// TIA Portal project "Projekt_skrzyzowanie_ZSP" (V13)

(* hardware
DEVICE "HMI_1"  KTP600 Basic color PN
   slot 0: "HMI"  HMI  6AV6 647-0AD11-3AX0  12.0.0.0
   slot 1: "HMI_RT_1"  KTP600 Basic color PN  6AV6 647-0AD11-3AX0  12.0.0.0
   slot 5: "HMI_1.IE_CP_1"  PROFINET Interface
      slot 1: "PROFINET Interface_1"  PROFINET Interface
         slot 1: "Port_1"  Port
DEVICE "S7-1200 station_2"  S7-1200 Station
   slot 0: "Rack_0"  Rack  V1.0
   slot 1: "PLC_1"  CPU 1212C AC/DC/Rly  6ES7 212-1BD30-0XB0  V2.2
*)

// ===== PLC "PLC_1"  CPU 1212C AC/DC/Rly =====

VAR_GLOBAL   // PLC tag table "Default tag table"
   "Clock_Byte" AT %MB0 : Byte;
   "Clock_10Hz" AT %M0.0 : Bool;
   "Clock_5Hz" AT %M0.1 : Bool;
   "Clock_2.5Hz" AT %M0.2 : Bool;
   "Clock_2Hz" AT %M0.3 : Bool;
   "Clock_1.25Hz" AT %M0.4 : Bool;
   "Clock_1Hz" AT %M0.5 : Bool;
   "Clock_0.625Hz" AT %M0.6 : Bool;
   "Clock_0.5Hz" AT %M0.7 : Bool;
END_VAR

VAR_GLOBAL   // PLC tag table "Tablica_wejsc"
   "przycisk_piesi_1" AT %M10.0 : Bool;
   "przycisk_piesi_2" AT %M10.1 : Bool;
   "przycisk_piesi_3" AT %M10.2 : Bool;
   "przycisk_piesi_4" AT %M10.3 : Bool;
   "przycisk_piesi_5" AT %M10.4 : Bool;
   "przycisk_piesi_6" AT %M10.5 : Bool;
   "petl_ind_czuj_1" AT %I0.0 : Bool;
   "petl_ind_czuj_2" AT %I0.1 : Bool;
   "petl_ind_czuj_3" AT %I0.2 : Bool;
   "petl_ind_czuj_5" AT %I0.3 : Bool;
   "petl_ind_czuj_6" AT %I0.4 : Bool;
   "petl_ind_czuj_8" AT %I0.5 : Bool;
   "petl_ind_czuj_9" AT %I0.6 : Bool;
   "przycisk_trybu_recznego" AT %I0.7 : Bool;
END_VAR

VAR_GLOBAL   // PLC tag table "Tablica_wyjsc"
   "sw_auto_z1" AT %M30.0 : Bool;
   "sw_auto_z2" AT %M30.1 : Bool;
   "sw_auto_z3" AT %M30.2 : Bool;
   "sw_auto_z4" AT %M30.3 : Bool;
   "sw_auto_z5" AT %M30.4 : Bool;
   "sw_auto_z6" AT %M30.5 : Bool;
   "sw_auto_z7" AT %M30.6 : Bool;
   "sw_auto_z8" AT %M30.7 : Bool;
   "sw_auto_z9" AT %M31.0 : Bool;
   "sw_auto_p1" AT %M31.1 : Bool;
   "sw_auto_p2" AT %M31.2 : Bool;
   "sw_auto_p3" AT %M31.3 : Bool;
   "sw_auto_p4" AT %M31.4 : Bool;
   "sw_auto_p5" AT %M31.5 : Bool;
   "sw_auto_p6" AT %M31.6 : Bool;
   "sw_auto_p7" AT %M31.7 : Bool;
   "sw_auto_p8" AT %M32.0 : Bool;
   "sw_auto_p9" AT %M32.1 : Bool;
   "sw_auto_c1" AT %M32.2 : Bool;
   "sw_auto_c2" AT %M32.3 : Bool;
   "sw_auto_c3" AT %M32.4 : Bool;
   "sw_auto_c4" AT %M32.5 : Bool;
   "sw_auto_c5" AT %M32.6 : Bool;
   "sw_auto_c6" AT %M32.7 : Bool;
   "sw_auto_c7" AT %M33.0 : Bool;
   "sw_auto_c8" AT %M33.1 : Bool;
   "sw_auto_c9" AT %M33.2 : Bool;
   "sw_piesi_z1" AT %M33.3 : Bool;
   "sw_piesi_z2" AT %M33.4 : Bool;
   "sw_piesi_z3" AT %M33.5 : Bool;
   "sw_piesi_z4" AT %M33.6 : Bool;
   "sw_piesi_z5" AT %M33.7 : Bool;
   "sw_piesi_z6" AT %M34.0 : Bool;
   "sw_piesi_c1" AT %M34.1 : Bool;
   "sw_piesi_c2" AT %M34.2 : Bool;
   "sw_piesi_c3" AT %M34.3 : Bool;
   "sw_piesi_c4" AT %M34.4 : Bool;
   "sw_piesi_c5" AT %M34.5 : Bool;
   "sw_piesi_c6" AT %M34.6 : Bool;
   "sw_tram_z1" AT %M34.7 : Bool;
   "sw_tram_z2" AT %M35.0 : Bool;
   "sw_tram_c1" AT %M35.1 : Bool;
   "sw_tram_c2" AT %M35.2 : Bool;
END_VAR

VAR_GLOBAL   // PLC tag table "Tablica_zmiennych_programowych"
   "krok_programu" AT %MW20 : Word;
   "tryb_sterowania_recznego" AT %M22.0 : Bool;
   "zmienna_piesi_1" AT %M22.1 : Bool;
   "zmienna_piesi_2" AT %M22.2 : Bool;
   "zmienna_piesi_3" AT %M22.3 : Bool;
   "zmienna_piesi_4" AT %M22.4 : Bool;
   "zmienna_piesi_5" AT %M22.5 : Bool;
   "zmienna_piesi_6" AT %M22.6 : Bool;
   "droga_prioryt_1" AT %M22.7 : Bool;
   "droga_prioryt_2" AT %M23.0 : Bool;
END_VAR

// folder: System blocks/Program resources

DATA_BLOCK "timer_sw_pom_krok_10"   // DB1
{ S7_Optimized_Access := 'FALSE' }
AUTHOR : Simatic
FAMILY : IEC
NAME : IEC_TMR
VERSION : 1.0
// stored: InstanceOfName ?
"?"
BEGIN
END_DATA_BLOCK

DATA_BLOCK "Timer_sw_ziel_krok_11"   // DB2
{ S7_Optimized_Access := 'FALSE' }
AUTHOR : Simatic
FAMILY : IEC
NAME : IEC_TMR
VERSION : 1.0
// stored: InstanceOfName ?
"?"
BEGIN
END_DATA_BLOCK

DATA_BLOCK "Timer_sw_pom_krok_12"   // DB3
{ S7_Optimized_Access := 'FALSE' }
AUTHOR : Simatic
FAMILY : IEC
NAME : IEC_TMR
VERSION : 1.0
// stored: InstanceOfName ?
"?"
BEGIN
END_DATA_BLOCK

DATA_BLOCK "Timer_drogi_priorytetowej_1"   // DB4
{ S7_Optimized_Access := 'FALSE' }
AUTHOR : Simatic
FAMILY : IEC
NAME : IEC_TMR
VERSION : 1.0
// stored: InstanceOfName ?
"?"
BEGIN
END_DATA_BLOCK

DATA_BLOCK "timer_sw_pom_krok_20"   // DB5
{ S7_Optimized_Access := 'FALSE' }
AUTHOR : Simatic
FAMILY : IEC
NAME : IEC_TMR
VERSION : 1.0
// stored: InstanceOfName ?
"?"
BEGIN
END_DATA_BLOCK

DATA_BLOCK "Timer_sw_ziel_krok_21"   // DB6
{ S7_Optimized_Access := 'FALSE' }
AUTHOR : Simatic
FAMILY : IEC
NAME : IEC_TMR
VERSION : 1.0
// stored: InstanceOfName ?
"?"
BEGIN
END_DATA_BLOCK

DATA_BLOCK "Timer_sw_pom_krok_22"   // DB7
{ S7_Optimized_Access := 'FALSE' }
AUTHOR : Simatic
FAMILY : IEC
NAME : IEC_TMR
VERSION : 1.0
// stored: InstanceOfName ?
"?"
BEGIN
END_DATA_BLOCK

DATA_BLOCK "timer_sw_pom_krok_30"   // DB8
{ S7_Optimized_Access := 'FALSE' }
AUTHOR : Simatic
FAMILY : IEC
NAME : IEC_TMR
VERSION : 1.0
// stored: InstanceOfName ?
"?"
BEGIN
END_DATA_BLOCK

DATA_BLOCK "Timer_sw_ziel_krok_31"   // DB9
{ S7_Optimized_Access := 'FALSE' }
AUTHOR : Simatic
FAMILY : IEC
NAME : IEC_TMR
VERSION : 1.0
// stored: InstanceOfName ?
"?"
BEGIN
END_DATA_BLOCK

DATA_BLOCK "Timer_sw_pom_krok_32"   // DB10
{ S7_Optimized_Access := 'FALSE' }
AUTHOR : Simatic
FAMILY : IEC
NAME : IEC_TMR
VERSION : 1.0
// stored: InstanceOfName ?
"?"
BEGIN
END_DATA_BLOCK

DATA_BLOCK "Timer_sw_czer_krok_33"   // DB11
{ S7_Optimized_Access := 'FALSE' }
AUTHOR : Simatic
FAMILY : IEC
NAME : IEC_TMR
VERSION : 1.0
// stored: InstanceOfName ?
"?"
BEGIN
END_DATA_BLOCK

DATA_BLOCK "Timer_sw_czer_krok_13"   // DB12
{ S7_Optimized_Access := 'FALSE' }
AUTHOR : Simatic
FAMILY : IEC
NAME : IEC_TMR
VERSION : 1.0
// stored: InstanceOfName ?
"?"
BEGIN
END_DATA_BLOCK

DATA_BLOCK "Timer_sw_czer_krok_23"   // DB13
{ S7_Optimized_Access := 'FALSE' }
AUTHOR : Simatic
FAMILY : IEC
NAME : IEC_TMR
VERSION : 1.0
// stored: InstanceOfName ?
"?"
BEGIN
END_DATA_BLOCK

DATA_BLOCK "timer_sw_pom_krok_40"   // DB14
{ S7_Optimized_Access := 'FALSE' }
AUTHOR : Simatic
FAMILY : IEC
NAME : IEC_TMR
VERSION : 1.0
// stored: InstanceOfName ?
"?"
BEGIN
END_DATA_BLOCK

DATA_BLOCK "Timer_sw_ziel_krok_41"   // DB15
{ S7_Optimized_Access := 'FALSE' }
AUTHOR : Simatic
FAMILY : IEC
NAME : IEC_TMR
VERSION : 1.0
// stored: InstanceOfName ?
"?"
BEGIN
END_DATA_BLOCK

DATA_BLOCK "Timer_sw_pom_krok_42"   // DB16
{ S7_Optimized_Access := 'FALSE' }
AUTHOR : Simatic
FAMILY : IEC
NAME : IEC_TMR
VERSION : 1.0
// stored: InstanceOfName ?
"?"
BEGIN
END_DATA_BLOCK

DATA_BLOCK "Timer_sw_czer_krok_43"   // DB17
{ S7_Optimized_Access := 'FALSE' }
AUTHOR : Simatic
FAMILY : IEC
NAME : IEC_TMR
VERSION : 1.0
// stored: InstanceOfName ?
"?"
BEGIN
END_DATA_BLOCK

DATA_BLOCK "1Timer_petli_ind_9"   // DB18
{ S7_Optimized_Access := 'FALSE' }
AUTHOR : Simatic
FAMILY : IEC
NAME : IEC_TMR
VERSION : 1.0
// stored: InstanceOfName ?
"?"
BEGIN
END_DATA_BLOCK

DATA_BLOCK "2Timer_petli_ind_9"   // DB19
{ S7_Optimized_Access := 'FALSE' }
AUTHOR : Simatic
FAMILY : IEC
NAME : IEC_TMR
VERSION : 1.0
// stored: InstanceOfName ?
"?"
BEGIN
END_DATA_BLOCK

DATA_BLOCK "Licznik_drog_prior2_1"   // DB20
{ S7_Optimized_Access := 'FALSE' }
AUTHOR : Simatic
FAMILY : IEC
NAME : CNTR
VERSION : 1.0
// stored: InstanceOfName ?
"?"
BEGIN
END_DATA_BLOCK

DATA_BLOCK "Licznik_drog_prior6_1"   // DB21
{ S7_Optimized_Access := 'FALSE' }
AUTHOR : Simatic
FAMILY : IEC
NAME : CNTR
VERSION : 1.0
// stored: InstanceOfName ?
"?"
BEGIN
END_DATA_BLOCK

DATA_BLOCK "Licznik_drog_prior1_2"   // DB22
{ S7_Optimized_Access := 'FALSE' }
AUTHOR : Simatic
FAMILY : IEC
NAME : CNTR
VERSION : 1.0
// stored: InstanceOfName ?
"?"
BEGIN
END_DATA_BLOCK

DATA_BLOCK "Licznik_drog_prior5_2"   // DB23
{ S7_Optimized_Access := 'FALSE' }
AUTHOR : Simatic
FAMILY : IEC
NAME : CNTR
VERSION : 1.0
// stored: InstanceOfName ?
"?"
BEGIN
END_DATA_BLOCK

DATA_BLOCK "Timer_drogi_priorytetowej_2"   // DB24
{ S7_Optimized_Access := 'FALSE' }
AUTHOR : Simatic
FAMILY : IEC
NAME : IEC_TMR
VERSION : 1.0
// stored: InstanceOfName ?
"?"
BEGIN
END_DATA_BLOCK

DATA_BLOCK "1Timer_zmiany_sw_piesi_1"   // DB25
{ S7_Optimized_Access := 'FALSE' }
AUTHOR : Simatic
FAMILY : IEC
NAME : IEC_TMR
VERSION : 1.0
// stored: InstanceOfName ?
"?"
BEGIN
END_DATA_BLOCK

DATA_BLOCK "1Timer_petli_ind_1"   // DB26
{ S7_Optimized_Access := 'FALSE' }
AUTHOR : Simatic
FAMILY : IEC
NAME : IEC_TMR
VERSION : 1.0
// stored: InstanceOfName ?
"?"
BEGIN
END_DATA_BLOCK

DATA_BLOCK "2Timer_petli_ind_1"   // DB27
{ S7_Optimized_Access := 'FALSE' }
AUTHOR : Simatic
FAMILY : IEC
NAME : IEC_TMR
VERSION : 1.0
// stored: InstanceOfName ?
"?"
BEGIN
END_DATA_BLOCK

DATA_BLOCK "1Timer_zmiany_sw_piesi_3"   // DB28
{ S7_Optimized_Access := 'FALSE' }
AUTHOR : Simatic
FAMILY : IEC
NAME : IEC_TMR
VERSION : 1.0
// stored: InstanceOfName ?
"?"
BEGIN
END_DATA_BLOCK

DATA_BLOCK "1Timer_petli_ind_3"   // DB29
{ S7_Optimized_Access := 'FALSE' }
AUTHOR : Simatic
FAMILY : IEC
NAME : IEC_TMR
VERSION : 1.0
// stored: InstanceOfName ?
"?"
BEGIN
END_DATA_BLOCK

DATA_BLOCK "2Timer_petli_ind_3"   // DB30
{ S7_Optimized_Access := 'FALSE' }
AUTHOR : Simatic
FAMILY : IEC
NAME : IEC_TMR
VERSION : 1.0
// stored: InstanceOfName ?
"?"
BEGIN
END_DATA_BLOCK

DATA_BLOCK "1Timer_zmiany_sw_piesi_4"   // DB31
{ S7_Optimized_Access := 'FALSE' }
AUTHOR : Simatic
FAMILY : IEC
NAME : IEC_TMR
VERSION : 1.0
// stored: InstanceOfName ?
"?"
BEGIN
END_DATA_BLOCK

DATA_BLOCK "1Timer_petli_ind_8"   // DB32
{ S7_Optimized_Access := 'FALSE' }
AUTHOR : Simatic
FAMILY : IEC
NAME : IEC_TMR
VERSION : 1.0
// stored: InstanceOfName ?
"?"
BEGIN
END_DATA_BLOCK

DATA_BLOCK "Timer_obsl_petl_ind_1"   // DB33
{ S7_Optimized_Access := 'FALSE' }
AUTHOR : Simatic
FAMILY : IEC
NAME : IEC_TMR
VERSION : 1.0
// stored: InstanceOfName ?
"?"
BEGIN
END_DATA_BLOCK

DATA_BLOCK "Timer_obsl_petl_ind_2"   // DB34
{ S7_Optimized_Access := 'FALSE' }
AUTHOR : Simatic
FAMILY : IEC
NAME : IEC_TMR
VERSION : 1.0
// stored: InstanceOfName ?
"?"
BEGIN
END_DATA_BLOCK

DATA_BLOCK "Timer_obsl_petl_ind_3"   // DB35
{ S7_Optimized_Access := 'FALSE' }
AUTHOR : Simatic
FAMILY : IEC
NAME : IEC_TMR
VERSION : 1.0
// stored: InstanceOfName ?
"?"
BEGIN
END_DATA_BLOCK

DATA_BLOCK "Timer_obsl_petl_ind_4"   // DB36
{ S7_Optimized_Access := 'FALSE' }
AUTHOR : Simatic
FAMILY : IEC
NAME : IEC_TMR
VERSION : 1.0
// stored: InstanceOfName ?
"?"
BEGIN
END_DATA_BLOCK

// folder: (top level)

FUNCTION "Algorytm_glowny" : Void   // FC1, LAD
{ S7_Optimized_Access := 'FALSE' }
VERSION : 0.1
   VAR_TEMP   // added for the SCL form of the ladder/FBD networks
      _w1 : Bool;
   END_VAR
BEGIN

REGION Network 1: Start programu
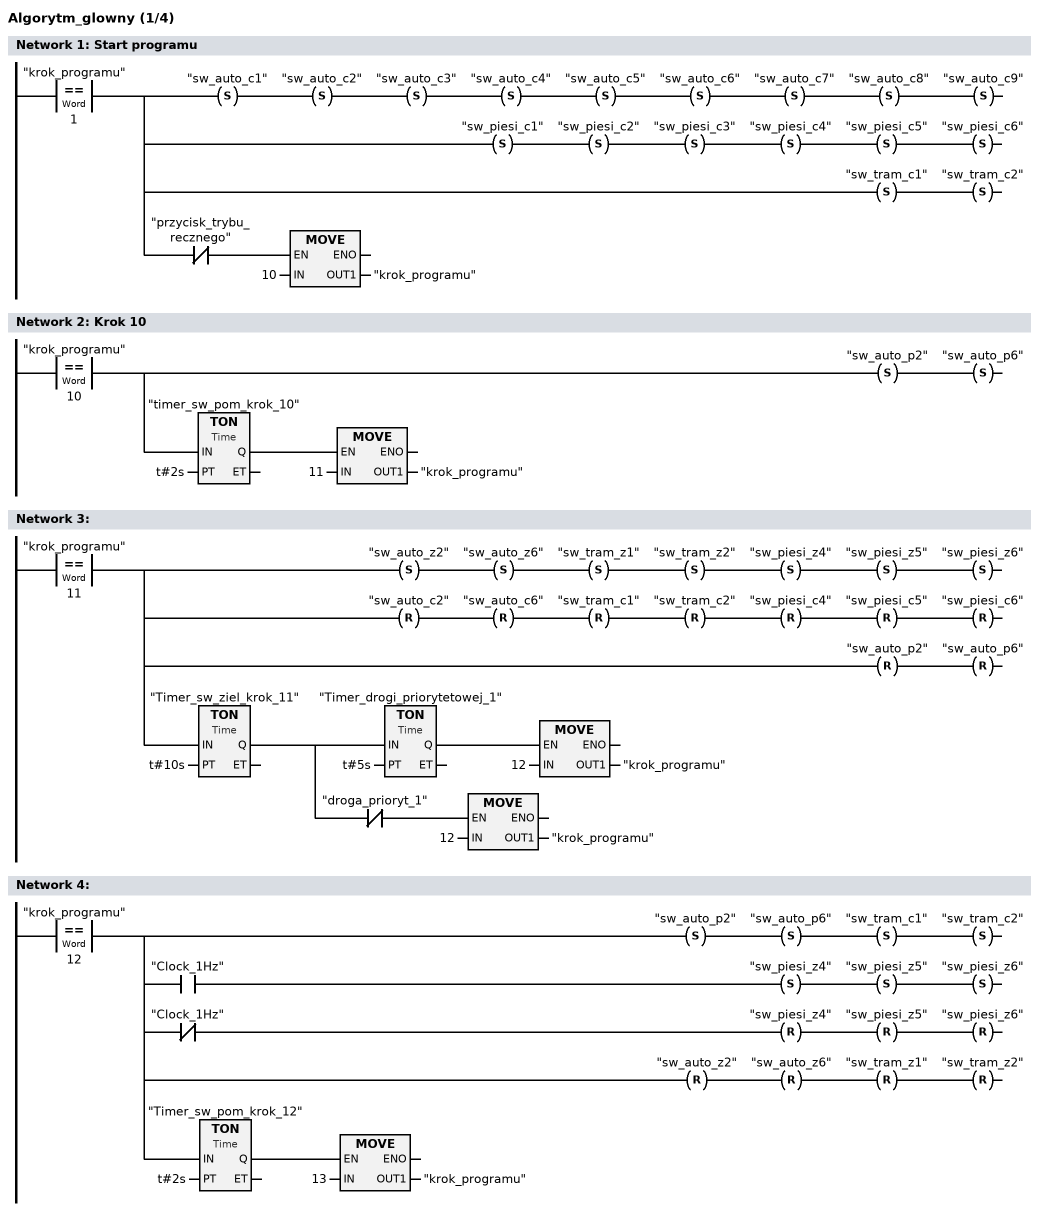
   RUNG wire#powerrail
      { S7_Templates := "SrcType := Word" } EQ_Contact(in1 := "krok_programu", in2 := 1)
      wire#w1
      S_Coil( "sw_auto_c1" )
      S_Coil( "sw_auto_c2" )
      S_Coil( "sw_auto_c3" )
      S_Coil( "sw_auto_c4" )
      S_Coil( "sw_auto_c5" )
      S_Coil( "sw_auto_c6" )
      S_Coil( "sw_auto_c7" )
      S_Coil( "sw_auto_c8" )
      S_Coil( "sw_auto_c9" )
   END_RUNG
   RUNG wire#w1
      S_Coil( "sw_piesi_c1" )
      S_Coil( "sw_piesi_c2" )
      S_Coil( "sw_piesi_c3" )
      S_Coil( "sw_piesi_c4" )
      S_Coil( "sw_piesi_c5" )
      S_Coil( "sw_piesi_c6" )
   END_RUNG
   RUNG wire#w1
      S_Coil( "sw_tram_c1" )
      S_Coil( "sw_tram_c2" )
   END_RUNG
   RUNG wire#w1
      I_Contact( "przycisk_trybu_recznego" )
      Move(in := 10, out1 => "krok_programu")
   END_RUNG
   // the same network as SCL:
   #_w1 := "krok_programu" = 1;
   IF #_w1 THEN
       "sw_auto_c1" := TRUE;
       "sw_auto_c2" := TRUE;
       "sw_auto_c3" := TRUE;
       "sw_auto_c4" := TRUE;
       "sw_auto_c5" := TRUE;
       "sw_auto_c6" := TRUE;
       "sw_auto_c7" := TRUE;
       "sw_auto_c8" := TRUE;
       "sw_auto_c9" := TRUE;
       "sw_piesi_c1" := TRUE;
       "sw_piesi_c2" := TRUE;
       "sw_piesi_c3" := TRUE;
       "sw_piesi_c4" := TRUE;
       "sw_piesi_c5" := TRUE;
       "sw_piesi_c6" := TRUE;
       "sw_tram_c1" := TRUE;
       "sw_tram_c2" := TRUE;
   END_IF;
   IF #_w1 AND NOT "przycisk_trybu_recznego" THEN "krok_programu" := 10; END_IF;
END_REGION

REGION Network 2: Krok 10
   #_w1 := "krok_programu" = 10;
   IF #_w1 THEN
       "sw_auto_p2" := TRUE;
       "sw_auto_p6" := TRUE;
   END_IF;
   "timer_sw_pom_krok_10".TON(IN := #_w1, PT := t#2s);
   IF "timer_sw_pom_krok_10".Q THEN "krok_programu" := 11; END_IF;
END_REGION

REGION Network 3
   #_w1 := "krok_programu" = 11;
   IF #_w1 THEN
       "sw_auto_z2" := TRUE;
       "sw_auto_z6" := TRUE;
       "sw_tram_z1" := TRUE;
       "sw_tram_z2" := TRUE;
       "sw_piesi_z4" := TRUE;
       "sw_piesi_z5" := TRUE;
       "sw_piesi_z6" := TRUE;
       "sw_auto_c2" := FALSE;
       "sw_auto_c6" := FALSE;
       "sw_tram_c1" := FALSE;
       "sw_tram_c2" := FALSE;
       "sw_piesi_c4" := FALSE;
       "sw_piesi_c5" := FALSE;
       "sw_piesi_c6" := FALSE;
       "sw_auto_p2" := FALSE;
       "sw_auto_p6" := FALSE;
   END_IF;
   "Timer_sw_ziel_krok_11".TON(IN := #_w1, PT := t#10s);
   "Timer_drogi_priorytetowej_1".TON(IN := "Timer_sw_ziel_krok_11".Q, PT := t#5s);
   IF "Timer_drogi_priorytetowej_1".Q THEN "krok_programu" := 12; END_IF;
   IF "Timer_sw_ziel_krok_11".Q AND NOT "droga_prioryt_1" THEN "krok_programu" := 12; END_IF;
END_REGION

REGION Network 4
   #_w1 := "krok_programu" = 12;
   IF #_w1 THEN
       "sw_auto_p2" := TRUE;
       "sw_auto_p6" := TRUE;
       "sw_tram_c1" := TRUE;
       "sw_tram_c2" := TRUE;
   END_IF;
   IF #_w1 AND "Clock_1Hz" THEN
       "sw_piesi_z4" := TRUE;
       "sw_piesi_z5" := TRUE;
       "sw_piesi_z6" := TRUE;
   END_IF;
   IF #_w1 AND NOT "Clock_1Hz" THEN
       "sw_piesi_z4" := FALSE;
       "sw_piesi_z5" := FALSE;
       "sw_piesi_z6" := FALSE;
   END_IF;
   IF #_w1 THEN
       "sw_auto_z2" := FALSE;
       "sw_auto_z6" := FALSE;
       "sw_tram_z1" := FALSE;
       "sw_tram_z2" := FALSE;
   END_IF;
   "Timer_sw_pom_krok_12".TON(IN := #_w1, PT := t#2s);
   IF "Timer_sw_pom_krok_12".Q THEN "krok_programu" := 13; END_IF;
END_REGION

REGION Network 5
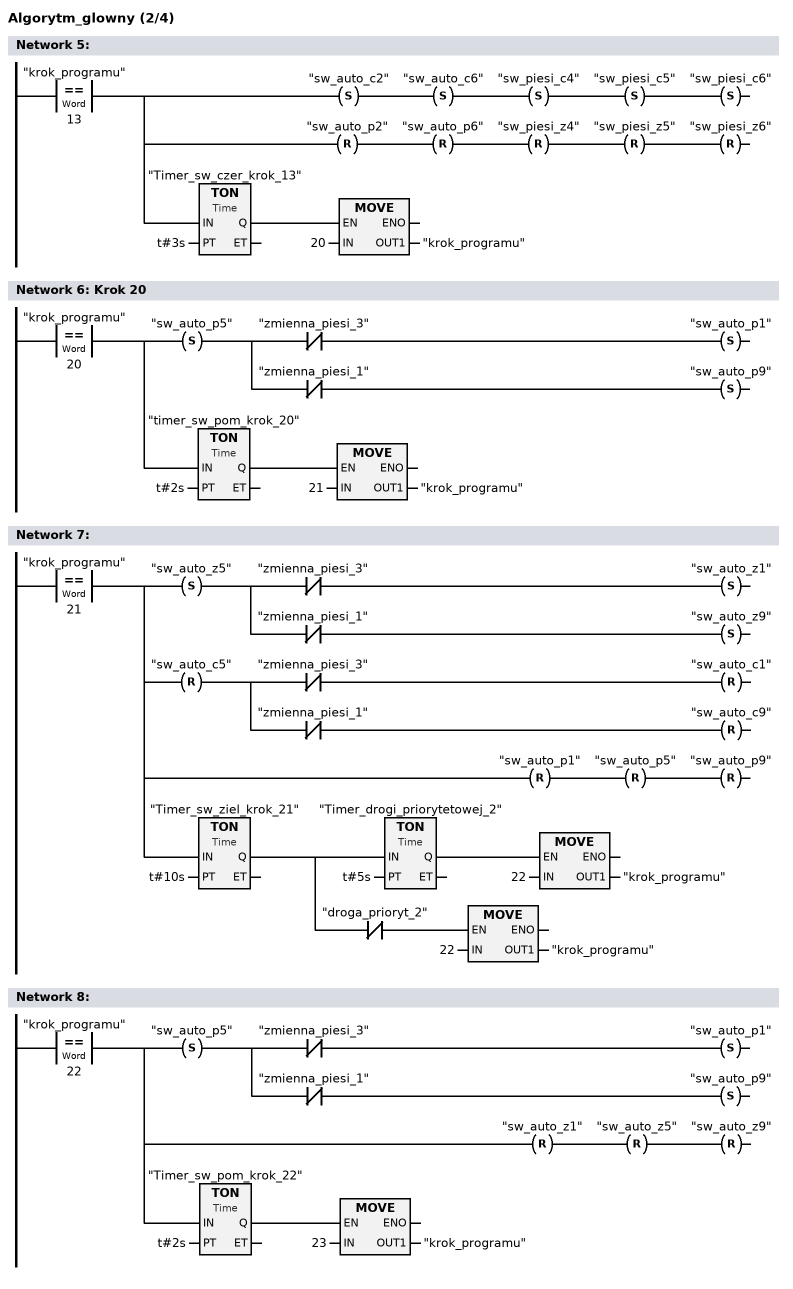
   #_w1 := "krok_programu" = 13;
   IF #_w1 THEN
       "sw_auto_c2" := TRUE;
       "sw_auto_c6" := TRUE;
       "sw_piesi_c4" := TRUE;
       "sw_piesi_c5" := TRUE;
       "sw_piesi_c6" := TRUE;
       "sw_auto_p2" := FALSE;
       "sw_auto_p6" := FALSE;
       "sw_piesi_z4" := FALSE;
       "sw_piesi_z5" := FALSE;
       "sw_piesi_z6" := FALSE;
   END_IF;
   "Timer_sw_czer_krok_13".TON(IN := #_w1, PT := t#3s);
   IF "Timer_sw_czer_krok_13".Q THEN "krok_programu" := 20; END_IF;
END_REGION

REGION Network 6: Krok 20
   #_w1 := "krok_programu" = 20;
   IF #_w1 THEN "sw_auto_p5" := TRUE; END_IF;
   IF #_w1 AND NOT "zmienna_piesi_3" THEN "sw_auto_p1" := TRUE; END_IF;
   IF #_w1 AND NOT "zmienna_piesi_1" THEN "sw_auto_p9" := TRUE; END_IF;
   "timer_sw_pom_krok_20".TON(IN := #_w1, PT := t#2s);
   IF "timer_sw_pom_krok_20".Q THEN "krok_programu" := 21; END_IF;
END_REGION

REGION Network 7
   #_w1 := "krok_programu" = 21;
   IF #_w1 THEN "sw_auto_z5" := TRUE; END_IF;
   IF #_w1 AND NOT "zmienna_piesi_3" THEN "sw_auto_z1" := TRUE; END_IF;
   IF #_w1 AND NOT "zmienna_piesi_1" THEN "sw_auto_z9" := TRUE; END_IF;
   IF #_w1 THEN "sw_auto_c5" := FALSE; END_IF;
   IF #_w1 AND NOT "zmienna_piesi_3" THEN "sw_auto_c1" := FALSE; END_IF;
   IF #_w1 AND NOT "zmienna_piesi_1" THEN "sw_auto_c9" := FALSE; END_IF;
   IF #_w1 THEN
       "sw_auto_p1" := FALSE;
       "sw_auto_p5" := FALSE;
       "sw_auto_p9" := FALSE;
   END_IF;
   "Timer_sw_ziel_krok_21".TON(IN := #_w1, PT := t#10s);
   "Timer_drogi_priorytetowej_2".TON(IN := "Timer_sw_ziel_krok_21".Q, PT := t#5s);
   IF "Timer_drogi_priorytetowej_2".Q THEN "krok_programu" := 22; END_IF;
   IF "Timer_sw_ziel_krok_21".Q AND NOT "droga_prioryt_2" THEN "krok_programu" := 22; END_IF;
END_REGION

REGION Network 8
   #_w1 := "krok_programu" = 22;
   IF #_w1 THEN "sw_auto_p5" := TRUE; END_IF;
   IF #_w1 AND NOT "zmienna_piesi_3" THEN "sw_auto_p1" := TRUE; END_IF;
   IF #_w1 AND NOT "zmienna_piesi_1" THEN "sw_auto_p9" := TRUE; END_IF;
   IF #_w1 THEN
       "sw_auto_z1" := FALSE;
       "sw_auto_z5" := FALSE;
       "sw_auto_z9" := FALSE;
   END_IF;
   "Timer_sw_pom_krok_22".TON(IN := #_w1, PT := t#2s);
   IF "Timer_sw_pom_krok_22".Q THEN "krok_programu" := 23; END_IF;
END_REGION

REGION Network 9
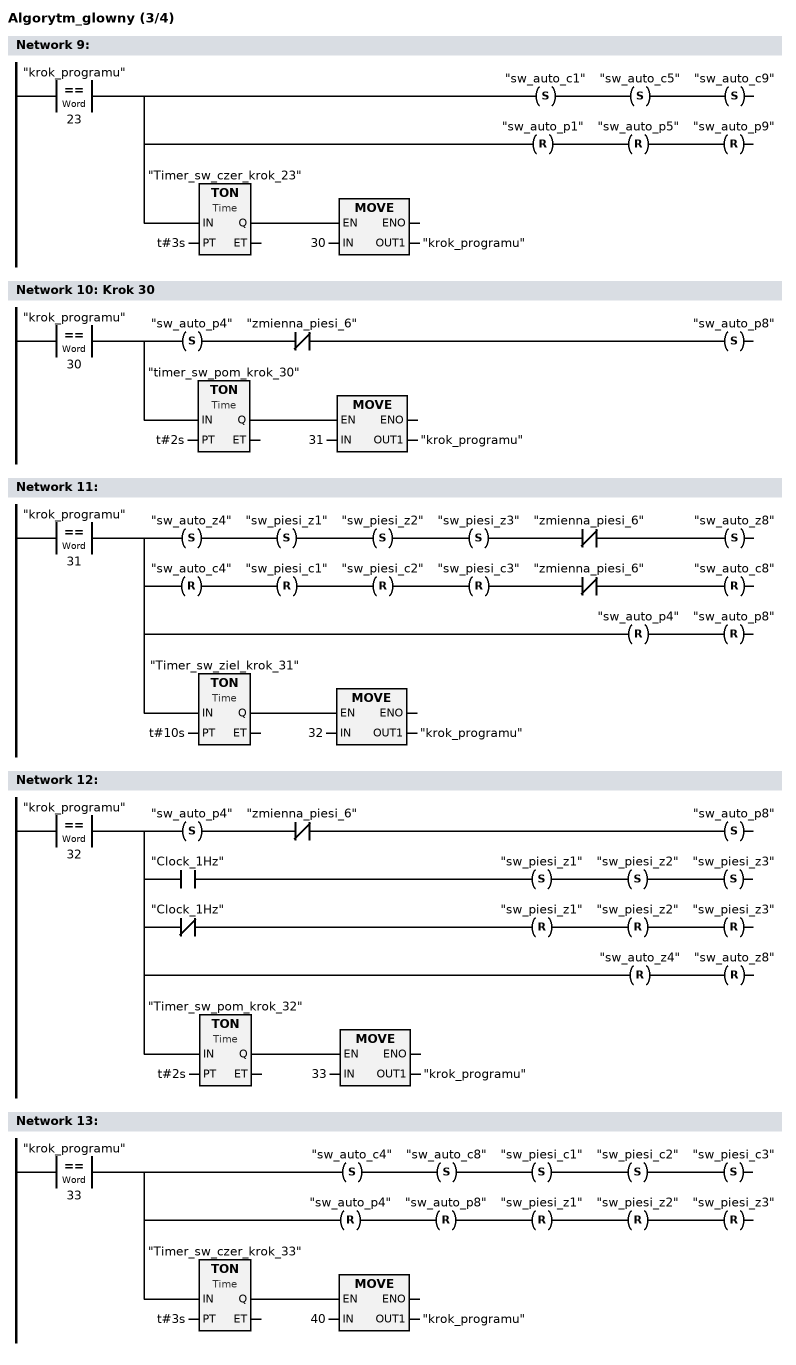
   #_w1 := "krok_programu" = 23;
   IF #_w1 THEN
       "sw_auto_c1" := TRUE;
       "sw_auto_c5" := TRUE;
       "sw_auto_c9" := TRUE;
       "sw_auto_p1" := FALSE;
       "sw_auto_p5" := FALSE;
       "sw_auto_p9" := FALSE;
   END_IF;
   "Timer_sw_czer_krok_23".TON(IN := #_w1, PT := t#3s);
   IF "Timer_sw_czer_krok_23".Q THEN "krok_programu" := 30; END_IF;
END_REGION

REGION Network 10: Krok 30
   #_w1 := "krok_programu" = 30;
   IF #_w1 THEN "sw_auto_p4" := TRUE; END_IF;
   IF #_w1 AND NOT "zmienna_piesi_6" THEN "sw_auto_p8" := TRUE; END_IF;
   "timer_sw_pom_krok_30".TON(IN := #_w1, PT := t#2s);
   IF "timer_sw_pom_krok_30".Q THEN "krok_programu" := 31; END_IF;
END_REGION

REGION Network 11
   #_w1 := "krok_programu" = 31;
   IF #_w1 THEN
       "sw_auto_z4" := TRUE;
       "sw_piesi_z1" := TRUE;
       "sw_piesi_z2" := TRUE;
       "sw_piesi_z3" := TRUE;
   END_IF;
   IF #_w1 AND NOT "zmienna_piesi_6" THEN "sw_auto_z8" := TRUE; END_IF;
   IF #_w1 THEN
       "sw_auto_c4" := FALSE;
       "sw_piesi_c1" := FALSE;
       "sw_piesi_c2" := FALSE;
       "sw_piesi_c3" := FALSE;
   END_IF;
   IF #_w1 AND NOT "zmienna_piesi_6" THEN "sw_auto_c8" := FALSE; END_IF;
   IF #_w1 THEN
       "sw_auto_p4" := FALSE;
       "sw_auto_p8" := FALSE;
   END_IF;
   "Timer_sw_ziel_krok_31".TON(IN := #_w1, PT := t#10s);
   IF "Timer_sw_ziel_krok_31".Q THEN "krok_programu" := 32; END_IF;
END_REGION

REGION Network 12
   #_w1 := "krok_programu" = 32;
   IF #_w1 THEN "sw_auto_p4" := TRUE; END_IF;
   IF #_w1 AND NOT "zmienna_piesi_6" THEN "sw_auto_p8" := TRUE; END_IF;
   IF #_w1 AND "Clock_1Hz" THEN
       "sw_piesi_z1" := TRUE;
       "sw_piesi_z2" := TRUE;
       "sw_piesi_z3" := TRUE;
   END_IF;
   IF #_w1 AND NOT "Clock_1Hz" THEN
       "sw_piesi_z1" := FALSE;
       "sw_piesi_z2" := FALSE;
       "sw_piesi_z3" := FALSE;
   END_IF;
   IF #_w1 THEN
       "sw_auto_z4" := FALSE;
       "sw_auto_z8" := FALSE;
   END_IF;
   "Timer_sw_pom_krok_32".TON(IN := #_w1, PT := t#2s);
   IF "Timer_sw_pom_krok_32".Q THEN "krok_programu" := 33; END_IF;
END_REGION

REGION Network 13
   #_w1 := "krok_programu" = 33;
   IF #_w1 THEN
       "sw_auto_c4" := TRUE;
       "sw_auto_c8" := TRUE;
       "sw_piesi_c1" := TRUE;
       "sw_piesi_c2" := TRUE;
       "sw_piesi_c3" := TRUE;
       "sw_auto_p4" := FALSE;
       "sw_auto_p8" := FALSE;
       "sw_piesi_z1" := FALSE;
       "sw_piesi_z2" := FALSE;
       "sw_piesi_z3" := FALSE;
   END_IF;
   "Timer_sw_czer_krok_33".TON(IN := #_w1, PT := t#3s);
   IF "Timer_sw_czer_krok_33".Q THEN "krok_programu" := 40; END_IF;
END_REGION

REGION Network 14: Krok 40
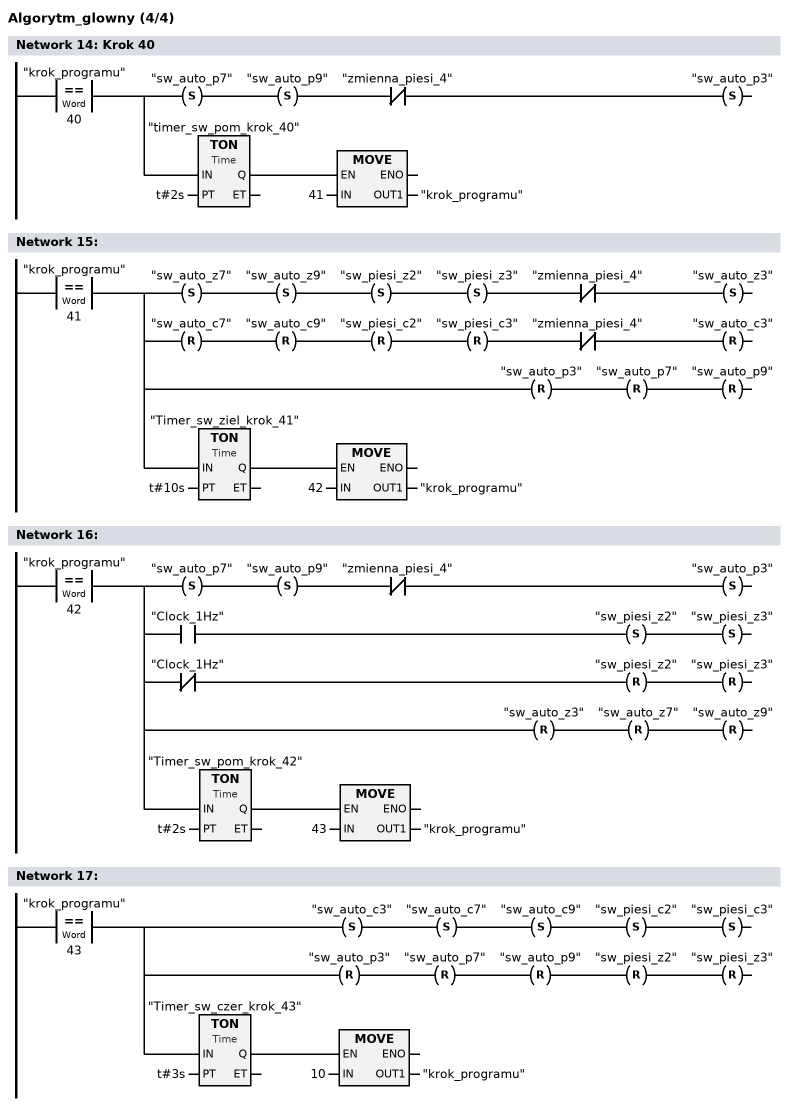
   #_w1 := "krok_programu" = 40;
   IF #_w1 THEN
       "sw_auto_p7" := TRUE;
       "sw_auto_p9" := TRUE;
   END_IF;
   IF #_w1 AND NOT "zmienna_piesi_4" THEN "sw_auto_p3" := TRUE; END_IF;
   "timer_sw_pom_krok_40".TON(IN := #_w1, PT := t#2s);
   IF "timer_sw_pom_krok_40".Q THEN "krok_programu" := 41; END_IF;
END_REGION

REGION Network 15
   #_w1 := "krok_programu" = 41;
   IF #_w1 THEN
       "sw_auto_z7" := TRUE;
       "sw_auto_z9" := TRUE;
       "sw_piesi_z2" := TRUE;
       "sw_piesi_z3" := TRUE;
   END_IF;
   IF #_w1 AND NOT "zmienna_piesi_4" THEN "sw_auto_z3" := TRUE; END_IF;
   IF #_w1 THEN
       "sw_auto_c7" := FALSE;
       "sw_auto_c9" := FALSE;
       "sw_piesi_c2" := FALSE;
       "sw_piesi_c3" := FALSE;
   END_IF;
   IF #_w1 AND NOT "zmienna_piesi_4" THEN "sw_auto_c3" := FALSE; END_IF;
   IF #_w1 THEN
       "sw_auto_p3" := FALSE;
       "sw_auto_p7" := FALSE;
       "sw_auto_p9" := FALSE;
   END_IF;
   "Timer_sw_ziel_krok_41".TON(IN := #_w1, PT := t#10s);
   IF "Timer_sw_ziel_krok_41".Q THEN "krok_programu" := 42; END_IF;
END_REGION

REGION Network 16
   #_w1 := "krok_programu" = 42;
   IF #_w1 THEN
       "sw_auto_p7" := TRUE;
       "sw_auto_p9" := TRUE;
   END_IF;
   IF #_w1 AND NOT "zmienna_piesi_4" THEN "sw_auto_p3" := TRUE; END_IF;
   IF #_w1 AND "Clock_1Hz" THEN
       "sw_piesi_z2" := TRUE;
       "sw_piesi_z3" := TRUE;
   END_IF;
   IF #_w1 AND NOT "Clock_1Hz" THEN
       "sw_piesi_z2" := FALSE;
       "sw_piesi_z3" := FALSE;
   END_IF;
   IF #_w1 THEN
       "sw_auto_z3" := FALSE;
       "sw_auto_z7" := FALSE;
       "sw_auto_z9" := FALSE;
   END_IF;
   "Timer_sw_pom_krok_42".TON(IN := #_w1, PT := t#2s);
   IF "Timer_sw_pom_krok_42".Q THEN "krok_programu" := 43; END_IF;
END_REGION

REGION Network 17
   #_w1 := "krok_programu" = 43;
   IF #_w1 THEN
       "sw_auto_c3" := TRUE;
       "sw_auto_c7" := TRUE;
       "sw_auto_c9" := TRUE;
       "sw_piesi_c2" := TRUE;
       "sw_piesi_c3" := TRUE;
       "sw_auto_p3" := FALSE;
       "sw_auto_p7" := FALSE;
       "sw_auto_p9" := FALSE;
       "sw_piesi_z2" := FALSE;
       "sw_piesi_z3" := FALSE;
   END_IF;
   "Timer_sw_czer_krok_43".TON(IN := #_w1, PT := t#3s);
   IF "Timer_sw_czer_krok_43".Q THEN "krok_programu" := 10; END_IF;
END_REGION
END_FUNCTION

FUNCTION "Sterowanie_reczne" : Void   // FC2, LAD
{ S7_Optimized_Access := 'FALSE' }
VERSION : 0.1
   VAR_TEMP   // added for the SCL form of the ladder/FBD networks
      _w1 : Bool;
   END_VAR
BEGIN

REGION Network 1
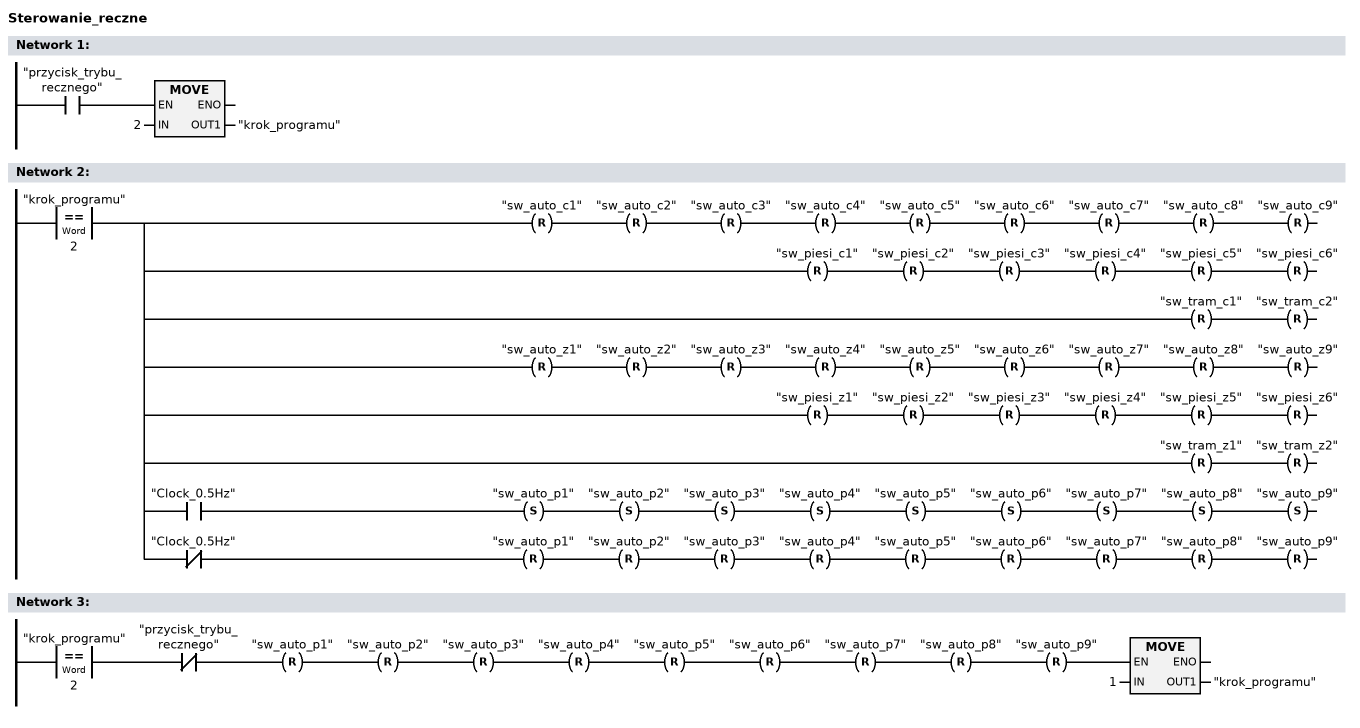
   RUNG wire#powerrail
      Contact( "przycisk_trybu_recznego" )
      Move(in := 2, out1 => "krok_programu")
   END_RUNG
   // the same network as SCL:
   IF "przycisk_trybu_recznego" THEN "krok_programu" := 2; END_IF;
END_REGION

REGION Network 2
   RUNG wire#powerrail
      { S7_Templates := "SrcType := Word" } EQ_Contact(in1 := "krok_programu", in2 := 2)
      wire#w1
      R_Coil( "sw_auto_c1" )
      R_Coil( "sw_auto_c2" )
      R_Coil( "sw_auto_c3" )
      R_Coil( "sw_auto_c4" )
      R_Coil( "sw_auto_c5" )
      R_Coil( "sw_auto_c6" )
      R_Coil( "sw_auto_c7" )
      R_Coil( "sw_auto_c8" )
      R_Coil( "sw_auto_c9" )
   END_RUNG
   RUNG wire#w1
      R_Coil( "sw_piesi_c1" )
      R_Coil( "sw_piesi_c2" )
      R_Coil( "sw_piesi_c3" )
      R_Coil( "sw_piesi_c4" )
      R_Coil( "sw_piesi_c5" )
      R_Coil( "sw_piesi_c6" )
   END_RUNG
   RUNG wire#w1
      R_Coil( "sw_tram_c1" )
      R_Coil( "sw_tram_c2" )
   END_RUNG
   RUNG wire#w1
      R_Coil( "sw_auto_z1" )
      R_Coil( "sw_auto_z2" )
      R_Coil( "sw_auto_z3" )
      R_Coil( "sw_auto_z4" )
      R_Coil( "sw_auto_z5" )
      R_Coil( "sw_auto_z6" )
      R_Coil( "sw_auto_z7" )
      R_Coil( "sw_auto_z8" )
      R_Coil( "sw_auto_z9" )
   END_RUNG
   RUNG wire#w1
      R_Coil( "sw_piesi_z1" )
      R_Coil( "sw_piesi_z2" )
      R_Coil( "sw_piesi_z3" )
      R_Coil( "sw_piesi_z4" )
      R_Coil( "sw_piesi_z5" )
      R_Coil( "sw_piesi_z6" )
   END_RUNG
   RUNG wire#w1
      R_Coil( "sw_tram_z1" )
      R_Coil( "sw_tram_z2" )
   END_RUNG
   RUNG wire#w1
      Contact( "Clock_0.5Hz" )
      S_Coil( "sw_auto_p1" )
      S_Coil( "sw_auto_p2" )
      S_Coil( "sw_auto_p3" )
      S_Coil( "sw_auto_p4" )
      S_Coil( "sw_auto_p5" )
      S_Coil( "sw_auto_p6" )
      S_Coil( "sw_auto_p7" )
      S_Coil( "sw_auto_p8" )
      S_Coil( "sw_auto_p9" )
   END_RUNG
   RUNG wire#w1
      I_Contact( "Clock_0.5Hz" )
      R_Coil( "sw_auto_p1" )
      R_Coil( "sw_auto_p2" )
      R_Coil( "sw_auto_p3" )
      R_Coil( "sw_auto_p4" )
      R_Coil( "sw_auto_p5" )
      R_Coil( "sw_auto_p6" )
      R_Coil( "sw_auto_p7" )
      R_Coil( "sw_auto_p8" )
      R_Coil( "sw_auto_p9" )
   END_RUNG
   // the same network as SCL:
   #_w1 := "krok_programu" = 2;
   IF #_w1 THEN
       "sw_auto_c1" := FALSE;
       "sw_auto_c2" := FALSE;
       "sw_auto_c3" := FALSE;
       "sw_auto_c4" := FALSE;
       "sw_auto_c5" := FALSE;
       "sw_auto_c6" := FALSE;
       "sw_auto_c7" := FALSE;
       "sw_auto_c8" := FALSE;
       "sw_auto_c9" := FALSE;
       "sw_piesi_c1" := FALSE;
       "sw_piesi_c2" := FALSE;
       "sw_piesi_c3" := FALSE;
       "sw_piesi_c4" := FALSE;
       "sw_piesi_c5" := FALSE;
       "sw_piesi_c6" := FALSE;
       "sw_tram_c1" := FALSE;
       "sw_tram_c2" := FALSE;
       "sw_auto_z1" := FALSE;
       "sw_auto_z2" := FALSE;
       "sw_auto_z3" := FALSE;
       "sw_auto_z4" := FALSE;
       "sw_auto_z5" := FALSE;
       "sw_auto_z6" := FALSE;
       "sw_auto_z7" := FALSE;
       "sw_auto_z8" := FALSE;
       "sw_auto_z9" := FALSE;
       "sw_piesi_z1" := FALSE;
       "sw_piesi_z2" := FALSE;
       "sw_piesi_z3" := FALSE;
       "sw_piesi_z4" := FALSE;
       "sw_piesi_z5" := FALSE;
       "sw_piesi_z6" := FALSE;
       "sw_tram_z1" := FALSE;
       "sw_tram_z2" := FALSE;
   END_IF;
   IF #_w1 AND "Clock_0.5Hz" THEN
       "sw_auto_p1" := TRUE;
       "sw_auto_p2" := TRUE;
       "sw_auto_p3" := TRUE;
       "sw_auto_p4" := TRUE;
       "sw_auto_p5" := TRUE;
       "sw_auto_p6" := TRUE;
       "sw_auto_p7" := TRUE;
       "sw_auto_p8" := TRUE;
       "sw_auto_p9" := TRUE;
   END_IF;
   IF #_w1 AND NOT "Clock_0.5Hz" THEN
       "sw_auto_p1" := FALSE;
       "sw_auto_p2" := FALSE;
       "sw_auto_p3" := FALSE;
       "sw_auto_p4" := FALSE;
       "sw_auto_p5" := FALSE;
       "sw_auto_p6" := FALSE;
       "sw_auto_p7" := FALSE;
       "sw_auto_p8" := FALSE;
       "sw_auto_p9" := FALSE;
   END_IF;
END_REGION

REGION Network 3
   RUNG wire#powerrail
      { S7_Templates := "SrcType := Word" } EQ_Contact(in1 := "krok_programu", in2 := 2)
      I_Contact( "przycisk_trybu_recznego" )
      R_Coil( "sw_auto_p1" )
      R_Coil( "sw_auto_p2" )
      R_Coil( "sw_auto_p3" )
      R_Coil( "sw_auto_p4" )
      R_Coil( "sw_auto_p5" )
      R_Coil( "sw_auto_p6" )
      R_Coil( "sw_auto_p7" )
      R_Coil( "sw_auto_p8" )
      R_Coil( "sw_auto_p9" )
      Move(in := 1, out1 => "krok_programu")
   END_RUNG
   // the same network as SCL:
   IF ("krok_programu" = 2) AND NOT "przycisk_trybu_recznego" THEN
       "sw_auto_p1" := FALSE;
       "sw_auto_p2" := FALSE;
       "sw_auto_p3" := FALSE;
       "sw_auto_p4" := FALSE;
       "sw_auto_p5" := FALSE;
       "sw_auto_p6" := FALSE;
       "sw_auto_p7" := FALSE;
       "sw_auto_p8" := FALSE;
       "sw_auto_p9" := FALSE;
       "krok_programu" := 1;
   END_IF;
END_REGION
END_FUNCTION

FUNCTION "Obsluga_drogi_priorytetowej" : Void   // FC3, LAD
{ S7_Optimized_Access := 'FALSE' }
VERSION : 0.1
BEGIN

REGION Network 1
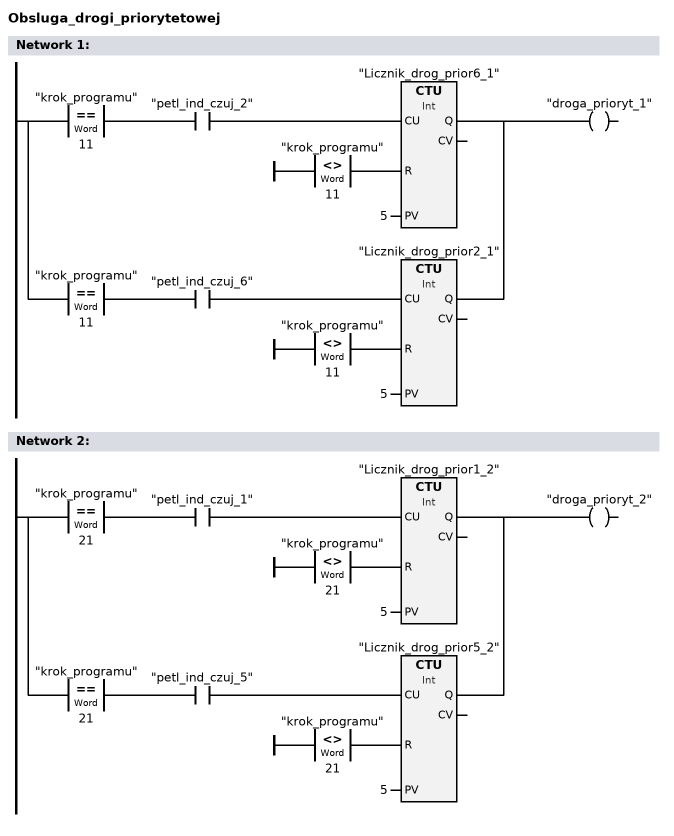
   "Licznik_drog_prior6_1".CTU(CU := ("krok_programu" = 11) AND "petl_ind_czuj_2",
                           R := "krok_programu" <> 11,
                           PV := 5);
   "Licznik_drog_prior2_1".CTU(CU := ("krok_programu" = 11) AND "petl_ind_czuj_6",
                           R := "krok_programu" <> 11,
                           PV := 5);
   "droga_prioryt_1" := "Licznik_drog_prior6_1".Q OR "Licznik_drog_prior2_1".Q;
END_REGION

REGION Network 2
   "Licznik_drog_prior1_2".CTU(CU := ("krok_programu" = 21) AND "petl_ind_czuj_1",
                           R := "krok_programu" <> 21,
                           PV := 5);
   "Licznik_drog_prior5_2".CTU(CU := ("krok_programu" = 21) AND "petl_ind_czuj_5",
                           R := "krok_programu" <> 21,
                           PV := 5);
   "droga_prioryt_2" := "Licznik_drog_prior1_2".Q OR "Licznik_drog_prior5_2".Q;
END_REGION
END_FUNCTION

FUNCTION "Przyciski_pieszych" : Void   // FC4, LAD
{ S7_Optimized_Access := 'FALSE' }
VERSION : 0.1
   VAR_TEMP   // added for the SCL form of the ladder/FBD networks
      _w1 : Bool;
   END_VAR
BEGIN

REGION Network 1: Piesi 1
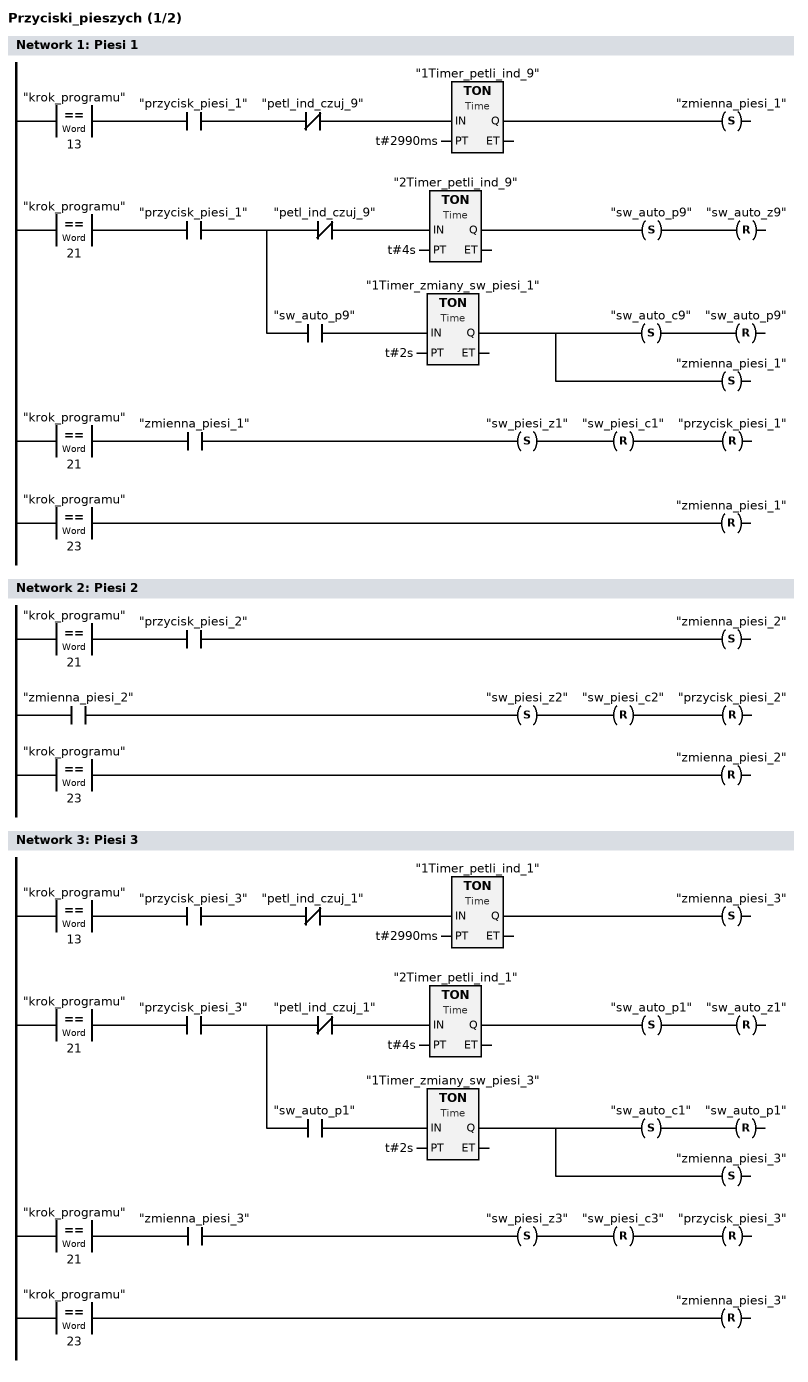
   "1Timer_petli_ind_9".TON(IN := ("krok_programu" = 13) AND "przycisk_piesi_1" AND NOT "petl_ind_czuj_9",
                           PT := t#2990ms);
   IF "1Timer_petli_ind_9".Q THEN "zmienna_piesi_1" := TRUE; END_IF;
   #_w1 := ("krok_programu" = 21) AND "przycisk_piesi_1";
   "2Timer_petli_ind_9".TON(IN := #_w1 AND NOT "petl_ind_czuj_9", PT := t#4s);
   IF "2Timer_petli_ind_9".Q THEN
       "sw_auto_p9" := TRUE;
       "sw_auto_z9" := FALSE;
   END_IF;
   "1Timer_zmiany_sw_piesi_1".TON(IN := #_w1 AND "sw_auto_p9", PT := t#2s);
   IF "1Timer_zmiany_sw_piesi_1".Q THEN
       "sw_auto_c9" := TRUE;
       "sw_auto_p9" := FALSE;
       "zmienna_piesi_1" := TRUE;
   END_IF;
   IF ("krok_programu" = 21) AND "zmienna_piesi_1" THEN
       "sw_piesi_z1" := TRUE;
       "sw_piesi_c1" := FALSE;
       "przycisk_piesi_1" := FALSE;
   END_IF;
   IF "krok_programu" = 23 THEN "zmienna_piesi_1" := FALSE; END_IF;
END_REGION

REGION Network 2: Piesi 2
   RUNG wire#powerrail
      { S7_Templates := "SrcType := Word" } EQ_Contact(in1 := "krok_programu", in2 := 21)
      Contact( "przycisk_piesi_2" )
      S_Coil( "zmienna_piesi_2" )
   END_RUNG
   RUNG wire#powerrail
      Contact( "zmienna_piesi_2" )
      S_Coil( "sw_piesi_z2" )
      R_Coil( "sw_piesi_c2" )
      R_Coil( "przycisk_piesi_2" )
   END_RUNG
   RUNG wire#powerrail
      { S7_Templates := "SrcType := Word" } EQ_Contact(in1 := "krok_programu", in2 := 23)
      R_Coil( "zmienna_piesi_2" )
   END_RUNG
   // the same network as SCL:
   IF ("krok_programu" = 21) AND "przycisk_piesi_2" THEN "zmienna_piesi_2" := TRUE; END_IF;
   IF "zmienna_piesi_2" THEN
       "sw_piesi_z2" := TRUE;
       "sw_piesi_c2" := FALSE;
       "przycisk_piesi_2" := FALSE;
   END_IF;
   IF "krok_programu" = 23 THEN "zmienna_piesi_2" := FALSE; END_IF;
END_REGION

REGION Network 3: Piesi 3
   "1Timer_petli_ind_1".TON(IN := ("krok_programu" = 13) AND "przycisk_piesi_3" AND NOT "petl_ind_czuj_1",
                           PT := t#2990ms);
   IF "1Timer_petli_ind_1".Q THEN "zmienna_piesi_3" := TRUE; END_IF;
   #_w1 := ("krok_programu" = 21) AND "przycisk_piesi_3";
   "2Timer_petli_ind_1".TON(IN := #_w1 AND NOT "petl_ind_czuj_1", PT := t#4s);
   IF "2Timer_petli_ind_1".Q THEN
       "sw_auto_p1" := TRUE;
       "sw_auto_z1" := FALSE;
   END_IF;
   "1Timer_zmiany_sw_piesi_3".TON(IN := #_w1 AND "sw_auto_p1", PT := t#2s);
   IF "1Timer_zmiany_sw_piesi_3".Q THEN
       "sw_auto_c1" := TRUE;
       "sw_auto_p1" := FALSE;
       "zmienna_piesi_3" := TRUE;
   END_IF;
   IF ("krok_programu" = 21) AND "zmienna_piesi_3" THEN
       "sw_piesi_z3" := TRUE;
       "sw_piesi_c3" := FALSE;
       "przycisk_piesi_3" := FALSE;
   END_IF;
   IF "krok_programu" = 23 THEN "zmienna_piesi_3" := FALSE; END_IF;
END_REGION

REGION Network 4: Piesi 4
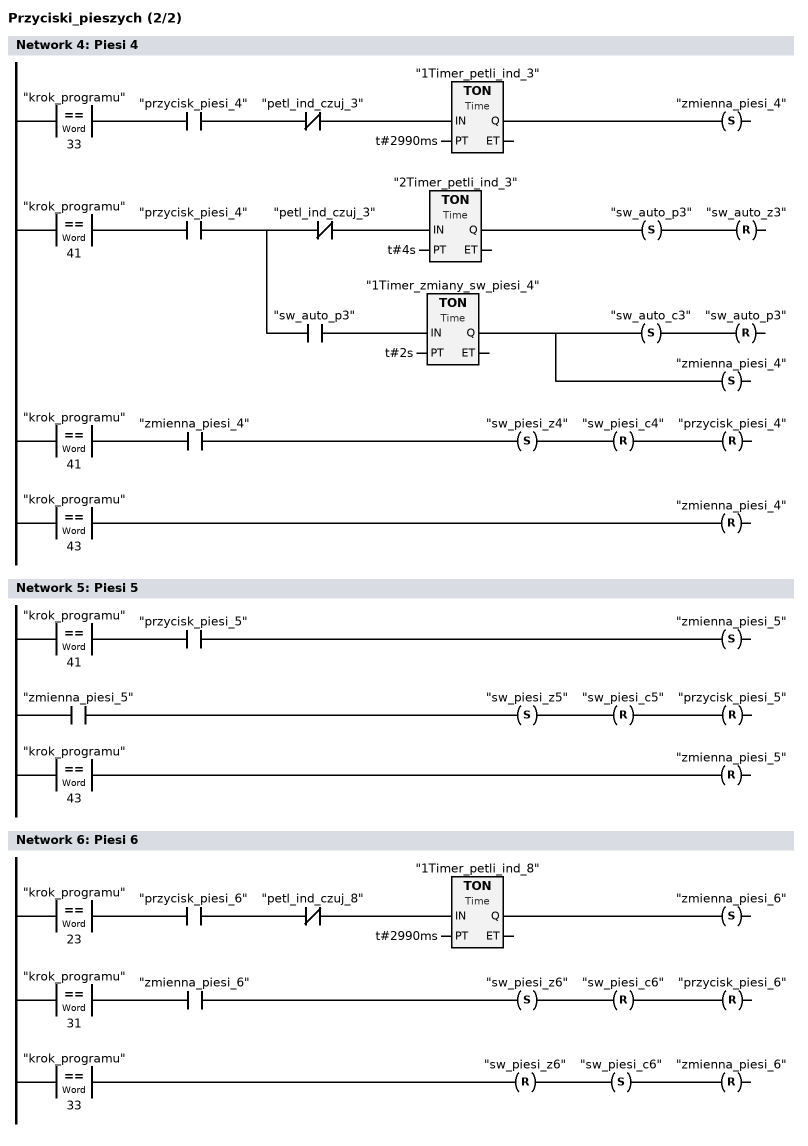
   "1Timer_petli_ind_3".TON(IN := ("krok_programu" = 33) AND "przycisk_piesi_4" AND NOT "petl_ind_czuj_3",
                           PT := t#2990ms);
   IF "1Timer_petli_ind_3".Q THEN "zmienna_piesi_4" := TRUE; END_IF;
   #_w1 := ("krok_programu" = 41) AND "przycisk_piesi_4";
   "2Timer_petli_ind_3".TON(IN := #_w1 AND NOT "petl_ind_czuj_3", PT := t#4s);
   IF "2Timer_petli_ind_3".Q THEN
       "sw_auto_p3" := TRUE;
       "sw_auto_z3" := FALSE;
   END_IF;
   "1Timer_zmiany_sw_piesi_4".TON(IN := #_w1 AND "sw_auto_p3", PT := t#2s);
   IF "1Timer_zmiany_sw_piesi_4".Q THEN
       "sw_auto_c3" := TRUE;
       "sw_auto_p3" := FALSE;
       "zmienna_piesi_4" := TRUE;
   END_IF;
   IF ("krok_programu" = 41) AND "zmienna_piesi_4" THEN
       "sw_piesi_z4" := TRUE;
       "sw_piesi_c4" := FALSE;
       "przycisk_piesi_4" := FALSE;
   END_IF;
   IF "krok_programu" = 43 THEN "zmienna_piesi_4" := FALSE; END_IF;
END_REGION

REGION Network 5: Piesi 5
   RUNG wire#powerrail
      { S7_Templates := "SrcType := Word" } EQ_Contact(in1 := "krok_programu", in2 := 41)
      Contact( "przycisk_piesi_5" )
      S_Coil( "zmienna_piesi_5" )
   END_RUNG
   RUNG wire#powerrail
      Contact( "zmienna_piesi_5" )
      S_Coil( "sw_piesi_z5" )
      R_Coil( "sw_piesi_c5" )
      R_Coil( "przycisk_piesi_5" )
   END_RUNG
   RUNG wire#powerrail
      { S7_Templates := "SrcType := Word" } EQ_Contact(in1 := "krok_programu", in2 := 43)
      R_Coil( "zmienna_piesi_5" )
   END_RUNG
   // the same network as SCL:
   IF ("krok_programu" = 41) AND "przycisk_piesi_5" THEN "zmienna_piesi_5" := TRUE; END_IF;
   IF "zmienna_piesi_5" THEN
       "sw_piesi_z5" := TRUE;
       "sw_piesi_c5" := FALSE;
       "przycisk_piesi_5" := FALSE;
   END_IF;
   IF "krok_programu" = 43 THEN "zmienna_piesi_5" := FALSE; END_IF;
END_REGION

REGION Network 6: Piesi 6
   "1Timer_petli_ind_8".TON(IN := ("krok_programu" = 23) AND "przycisk_piesi_6" AND NOT "petl_ind_czuj_8",
                           PT := t#2990ms);
   IF "1Timer_petli_ind_8".Q THEN "zmienna_piesi_6" := TRUE; END_IF;
   IF ("krok_programu" = 31) AND "zmienna_piesi_6" THEN
       "sw_piesi_z6" := TRUE;
       "sw_piesi_c6" := FALSE;
       "przycisk_piesi_6" := FALSE;
   END_IF;
   IF "krok_programu" = 33 THEN
       "sw_piesi_z6" := FALSE;
       "sw_piesi_c6" := TRUE;
       "zmienna_piesi_6" := FALSE;
   END_IF;
END_REGION
END_FUNCTION

FUNCTION "Obsluga_petli_indukcyjnych" : Void   // FC5, LAD
{ S7_Optimized_Access := 'FALSE' }
VERSION : 0.1
BEGIN

REGION Network 1: Obsluga dla kroku 13
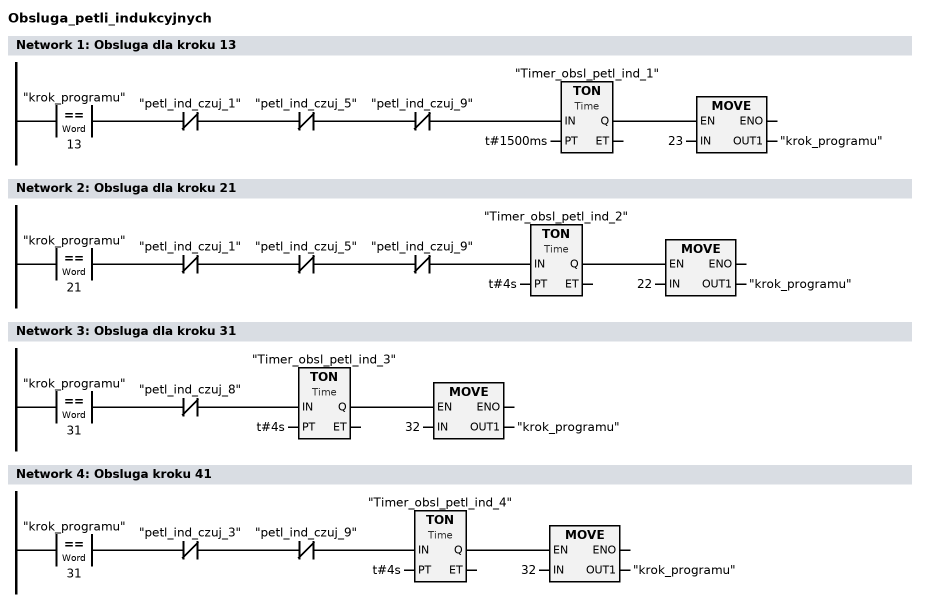
   "Timer_obsl_petl_ind_1".TON(IN := ("krok_programu" = 13) AND NOT "petl_ind_czuj_1" AND NOT "petl_ind_czuj_5" AND NOT "petl_ind_czuj_9",
                           PT := t#1500ms);
   IF "Timer_obsl_petl_ind_1".Q THEN "krok_programu" := 23; END_IF;
END_REGION

REGION Network 2: Obsluga dla kroku 21
   "Timer_obsl_petl_ind_2".TON(IN := ("krok_programu" = 21) AND NOT "petl_ind_czuj_1" AND NOT "petl_ind_czuj_5" AND NOT "petl_ind_czuj_9",
                           PT := t#4s);
   IF "Timer_obsl_petl_ind_2".Q THEN "krok_programu" := 22; END_IF;
END_REGION

REGION Network 3: Obsluga dla kroku 31
   "Timer_obsl_petl_ind_3".TON(IN := ("krok_programu" = 31) AND NOT "petl_ind_czuj_8", PT := t#4s);
   IF "Timer_obsl_petl_ind_3".Q THEN "krok_programu" := 32; END_IF;
END_REGION

REGION Network 4: Obsluga kroku 41
   "Timer_obsl_petl_ind_4".TON(IN := ("krok_programu" = 31) AND NOT "petl_ind_czuj_3" AND NOT "petl_ind_czuj_9",
                           PT := t#4s);
   IF "Timer_obsl_petl_ind_4".Q THEN "krok_programu" := 32; END_IF;
END_REGION
END_FUNCTION

ORGANIZATION_BLOCK "Main"   // OB1, LAD, ProgramCycle
TITLE = "Main Program Sweep (Cycle)"
{ S7_Optimized_Access := 'FALSE' }
VERSION : 0.1
   VAR_TEMP   // added for the SCL form of the ladder/FBD networks
      _w1 : Bool;
      _w2 : Bool;
      _w3 : Bool;
   END_VAR
BEGIN

REGION Network 1
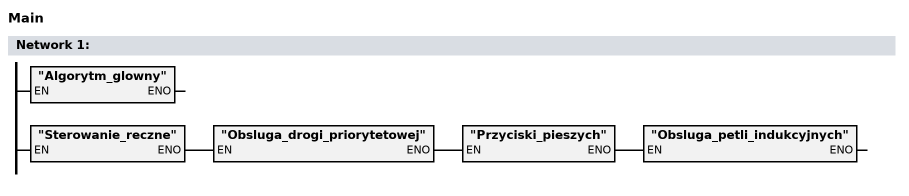
   RUNG wire#powerrail
      "Algorytm_glowny"()
   END_RUNG
   RUNG wire#powerrail
      "Sterowanie_reczne"()
      "Obsluga_drogi_priorytetowej"()
      "Przyciski_pieszych"()
      "Obsluga_petli_indukcyjnych"()
   END_RUNG
   // the same network as SCL:
   "Algorytm_glowny"();
   "Sterowanie_reczne"(ENO => #_w1);
   "Obsluga_drogi_priorytetowej"(EN := #_w1, ENO => #_w2);
   "Przyciski_pieszych"(EN := #_w2, ENO => #_w3);
   IF #_w3 THEN "Obsluga_petli_indukcyjnych"(); END_IF;
END_REGION
END_ORGANIZATION_BLOCK